Staubli VAL3: PROG.dtx

public progItem pProg{}
  [HOME1]
    InstrItem iEvent
      [0]
        string sType
        string sData
    string sID = "HOME1"
  [HOME2]
    InstrItem iEvent
      [0]
        string sType
        string sData
    string sID = "HOME2"
